FUNCTION angSpdCommandLimiter : LREAL
VAR_INPUT
	angSpdCommand:LREAL;
END_VAR
VAR
angRate:lreal;
END_VAR

angRate := (angSpdCommand - angSpdCommandShaped)/PLC_CYCLE;

  IF (ANGSPDRATELIMIT < angRate)THEN
    angRate := ANGSPDRATELIMIT;
  END_IF

  IF (-1*ANGSPDRATELIMIT > angRate)THEN
    angRate := -1 * ANGSPDRATELIMIT;
  END_IF

angSpdCommandShaped := angSpdCommandShaped+angRate * PLC_CYCLE;

IF(angSpdCommandShaped >= 40) THEN
 angSpdCommandShaped := 40;
 END_IF
IF(angSpdCommandShaped <= -40) THEN
 angSpdCommandShaped:= -40;
 END_IF
 angSpdCommandLimiter:=0;

END_FUNCTION

(* stored: Version 1.1.0.1, ProductVersion 3.1.4024.12
   POU angSpdCommandLimiter: Id {99b656ea-f8b3-409a-b618-aee19afa2417}, SpecialFunc None *)
